(* IEC 61131-3 sources: AXOpen/src/_test/app/SystemConstants, 2 files *)

(* ---- plc_line_IoAddresses.st ---- *)
CONFIGURATION IoAddresses
    VAR_GLOBAL

        // Module rexroth_ctrlx_drive/Inputs
        rexroth_ctrlx_drive_Inputs_P_0_0106_0_0__STO_function__Operating_status_Input AT %IB20 : rexroth_ctrlx_drive_Inputs_P_0_0106_0_0__STO_function__Operating_status_Input_Layout;
        rexroth_ctrlx_drive_Inputs_S_0_0084_0_0__Torque_force_feedback_value_Input AT %IB18 : rexroth_ctrlx_drive_Inputs_S_0_0084_0_0__Torque_force_feedback_value_Input_Layout;
        rexroth_ctrlx_drive_Inputs_S_0_0135_0_0__Drive_status_word__Value_Input AT %IB12 : rexroth_ctrlx_drive_Inputs_S_0_0135_0_0__Drive_status_word__Value_Input_Layout;
        rexroth_ctrlx_drive_Inputs_S_0_0144_0_0__Signal_status_word__Value_Input AT %IB14 : rexroth_ctrlx_drive_Inputs_S_0_0144_0_0__Signal_status_word__Value_Input_Layout;
        rexroth_ctrlx_drive_Inputs_S_0_0386_0_0__Position_controller__Position_actual_value_Input AT %IB0 : rexroth_ctrlx_drive_Inputs_S_0_0386_0_0__Position_controller__Position_actual_value_Input_Layout;
        rexroth_ctrlx_drive_Inputs_S_0_0390_0_0__Diagnostic_message__Manufacturer_status_register_Input AT %IB8 : rexroth_ctrlx_drive_Inputs_S_0_0390_0_0__Diagnostic_message__Manufacturer_status_register_Input_Layout;
        rexroth_ctrlx_drive_Inputs_S_0_0535_0_0__Velocity_controller__Velocity_actual_value_Input AT %IB4 : rexroth_ctrlx_drive_Inputs_S_0_0535_0_0__Velocity_controller__Velocity_actual_value_Input_Layout;
        rexroth_ctrlx_drive_Inputs_S_0_1720_0_2__Power_supply_control__Status_word_Input AT %IB16 : rexroth_ctrlx_drive_Inputs_S_0_1720_0_2__Power_supply_control__Status_word_Input_Layout;

        // Module rexroth_ctrlx_drive/Outputs
        rexroth_ctrlx_drive_Outputs_S_0_0080_0_0__Torque_force_command_value_Output AT %QB24 : rexroth_ctrlx_drive_Outputs_S_0_0080_0_0__Torque_force_command_value_Output_Layout;
        rexroth_ctrlx_drive_Outputs_S_0_0092_0_0__Torque_force_limitation__Limit_value_bipolar_Output AT %QB22 : rexroth_ctrlx_drive_Outputs_S_0_0092_0_0__Torque_force_limitation__Limit_value_bipolar_Output_Layout;
        rexroth_ctrlx_drive_Outputs_S_0_0134_0_0__Master_control_word__Value_Output AT %QB0 : rexroth_ctrlx_drive_Outputs_S_0_0134_0_0__Master_control_word__Value_Output_Layout;
        rexroth_ctrlx_drive_Outputs_S_0_0145_0_0__Signal_control_word__Value_Output AT %QB18 : rexroth_ctrlx_drive_Outputs_S_0_0145_0_0__Signal_control_word__Value_Output_Layout;
        rexroth_ctrlx_drive_Outputs_S_0_0193_0_0__Positioning_jerk_Output AT %QB26 : rexroth_ctrlx_drive_Outputs_S_0_0193_0_0__Positioning_jerk_Output_Layout;
        rexroth_ctrlx_drive_Outputs_S_0_0259_0_0__Positioning_profile__Profile_velocity_Output AT %QB14 : rexroth_ctrlx_drive_Outputs_S_0_0259_0_0__Positioning_profile__Profile_velocity_Output_Layout;
        rexroth_ctrlx_drive_Outputs_S_0_0260_0_0__Positioning_profile__Acceleration_Output AT %QB2 : rexroth_ctrlx_drive_Outputs_S_0_0260_0_0__Positioning_profile__Acceleration_Output_Layout;
        rexroth_ctrlx_drive_Outputs_S_0_0282_0_0__Drive_controlled_positioning__Command_value_Output AT %QB6 : rexroth_ctrlx_drive_Outputs_S_0_0282_0_0__Drive_controlled_positioning__Command_value_Output_Layout;
        rexroth_ctrlx_drive_Outputs_S_0_0359_0_0__Positioning_profile__Deceleration_Output AT %QB10 : rexroth_ctrlx_drive_Outputs_S_0_0359_0_0__Positioning_profile__Deceleration_Output_Layout;
        rexroth_ctrlx_drive_Outputs_S_0_1720_0_1__Power_supply_control__Control_word_Output AT %QB20 : rexroth_ctrlx_drive_Outputs_S_0_1720_0_1__Power_supply_control__Control_word_Output_Layout;
    END_VAR
END_CONFIGURATION

TYPE
    rexroth_ctrlx_drive_Inputs_P_0_0106_0_0__STO_function__Operating_status_Input_Layout : STRUCT
        Signals_0 AT %B0 : WORD;
    END_STRUCT;
END_TYPE

TYPE
    rexroth_ctrlx_drive_Inputs_S_0_0084_0_0__Torque_force_feedback_value_Input_Layout : STRUCT
        Signals_0 AT %B0 : INT;
    END_STRUCT;
END_TYPE

TYPE
    rexroth_ctrlx_drive_Inputs_S_0_0135_0_0__Drive_status_word__Value_Input_Layout : STRUCT
        Signals_0 AT %X0.3 : BOOL;
        Signals_1 AT %X0.4 : BOOL;
        Signals_2 AT %X0.5 : BOOL;
        Signals_3 AT %X0.7 : BOOL;
        Signals_4 AT %X1.0 : BOOL;
        Signals_5 AT %X1.1 : BOOL;
        Signals_6 AT %X1.2 : BOOL;
        Signals_7 AT %X1.4 : BOOL;
        Signals_8 AT %X1.5 : BOOL;
        Signals_9 AT %X1.6 : BOOL;
        Signals_10 AT %X1.7 : BOOL;
    END_STRUCT;
END_TYPE

TYPE
    rexroth_ctrlx_drive_Inputs_S_0_0144_0_0__Signal_status_word__Value_Input_Layout : STRUCT
        Signals_0 AT %B0 : WORD;
    END_STRUCT;
END_TYPE

TYPE
    rexroth_ctrlx_drive_Inputs_S_0_0386_0_0__Position_controller__Position_actual_value_Input_Layout : STRUCT
        Signals_0 AT %B0 : DINT;
    END_STRUCT;
END_TYPE

TYPE
    rexroth_ctrlx_drive_Inputs_S_0_0390_0_0__Diagnostic_message__Manufacturer_status_register_Input_Layout : STRUCT
        Signals_0 AT %B0 : DWORD;
    END_STRUCT;
END_TYPE

TYPE
    rexroth_ctrlx_drive_Inputs_S_0_0535_0_0__Velocity_controller__Velocity_actual_value_Input_Layout : STRUCT
        Signals_0 AT %B0 : DINT;
    END_STRUCT;
END_TYPE

TYPE
    rexroth_ctrlx_drive_Inputs_S_0_1720_0_2__Power_supply_control__Status_word_Input_Layout : STRUCT
        Signals_0 AT %B0 : WORD;
    END_STRUCT;
END_TYPE

TYPE
    rexroth_ctrlx_drive_Outputs_S_0_0080_0_0__Torque_force_command_value_Output_Layout : STRUCT
        Signals_0 AT %B0 : INT;
    END_STRUCT;
END_TYPE

TYPE
    rexroth_ctrlx_drive_Outputs_S_0_0092_0_0__Torque_force_limitation__Limit_value_bipolar_Output_Layout : STRUCT
        Signals_0 AT %B0 : WORD;
    END_STRUCT;
END_TYPE

TYPE
    rexroth_ctrlx_drive_Outputs_S_0_0134_0_0__Master_control_word__Value_Output_Layout : STRUCT
        Signals_0 AT %X1.0 : BOOL;
        Signals_1 AT %X1.1 : BOOL;
        Signals_2 AT %X1.2 : BOOL;
        Signals_3 AT %X1.5 : BOOL;
        Signals_4 AT %X1.6 : BOOL;
        Signals_5 AT %X1.7 : BOOL;
    END_STRUCT;
END_TYPE

TYPE
    rexroth_ctrlx_drive_Outputs_S_0_0145_0_0__Signal_control_word__Value_Output_Layout : STRUCT
        Signals_0 AT %B0 : WORD;
    END_STRUCT;
END_TYPE

TYPE
    rexroth_ctrlx_drive_Outputs_S_0_0193_0_0__Positioning_jerk_Output_Layout : STRUCT
        Signals_0 AT %B0 : DINT;
    END_STRUCT;
END_TYPE

TYPE
    rexroth_ctrlx_drive_Outputs_S_0_0259_0_0__Positioning_profile__Profile_velocity_Output_Layout : STRUCT
        Signals_0 AT %B0 : DWORD;
    END_STRUCT;
END_TYPE

TYPE
    rexroth_ctrlx_drive_Outputs_S_0_0260_0_0__Positioning_profile__Acceleration_Output_Layout : STRUCT
        Signals_0 AT %B0 : DINT;
    END_STRUCT;
END_TYPE

TYPE
    rexroth_ctrlx_drive_Outputs_S_0_0282_0_0__Drive_controlled_positioning__Command_value_Output_Layout : STRUCT
        Signals_0 AT %B0 : DINT;
    END_STRUCT;
END_TYPE

TYPE
    rexroth_ctrlx_drive_Outputs_S_0_0359_0_0__Positioning_profile__Deceleration_Output_Layout : STRUCT
        Signals_0 AT %B0 : DINT;
    END_STRUCT;
END_TYPE

TYPE
    rexroth_ctrlx_drive_Outputs_S_0_1720_0_1__Power_supply_control__Control_word_Output_Layout : STRUCT
        Signals_0 AT %B0 : WORD;
    END_STRUCT;
END_TYPE

(* ---- plc_line_HwIdentifiers.st ---- *)
CONFIGURATION HardwareIDs
    VAR_GLOBAL CONSTANT
        plc_line_HwID : UINT := UINT#32;
        plc_line_Rail_0_HwID : UINT := UINT#284;
        plc_line_plc_line_HwID : UINT := UINT#48;
        plc_line_plc_line_CPU_display_1_HwID : UINT := UINT#54;
        plc_line_plc_line_Card_reader_writer_1_HwID : UINT := UINT#51;
        plc_line_plc_line_DP_interface_1_HwID : UINT := UINT#60;
        plc_line_plc_line_OPC_UA_1_HwID : UINT := UINT#117;
        plc_line_plc_line_PROFINET_interface_1_HwID : UINT := UINT#64;
        plc_line_plc_line_PROFINET_interface_1_Port_1_HwID : UINT := UINT#65;
        plc_line_plc_line_PROFINET_interface_1_Port_2_HwID : UINT := UINT#66;
        plc_line_plc_line_PROFINET_interface_2_HwID : UINT := UINT#72;
        plc_line_plc_line_PROFINET_interface_2_Port_3_HwID : UINT := UINT#73;
        plc_line_plc_line_Virtual_communication_interface_HwID : UINT := UINT#135;
        profinet_plc_line_HwID : UINT := UINT#256;
        rexroth_ctrlx_drive_HwID : UINT := UINT#258;
        rexroth_ctrlx_drive_Inputs_HwID : UINT := UINT#264;
        rexroth_ctrlx_drive_Outputs_HwID : UINT := UINT#263;
        rexroth_ctrlx_drive_P_0_0106_0_0__STO_function__Operating_status_HwID : UINT := UINT#272;
        rexroth_ctrlx_drive_Rack_HwID : UINT := UINT#261;
        rexroth_ctrlx_drive_S_0_0080_0_0__Torque_force_command_value_HwID : UINT := UINT#281;
        rexroth_ctrlx_drive_S_0_0084_0_0__Torque_force_feedback_value_HwID : UINT := UINT#271;
        rexroth_ctrlx_drive_S_0_0092_0_0__Torque_force_limitation__Limit_value_bipolar_HwID : UINT := UINT#280;
        rexroth_ctrlx_drive_S_0_0134_0_0__Master_control_word__Value_HwID : UINT := UINT#273;
        rexroth_ctrlx_drive_S_0_0135_0_0__Drive_status_word__Value_HwID : UINT := UINT#268;
        rexroth_ctrlx_drive_S_0_0144_0_0__Signal_status_word__Value_HwID : UINT := UINT#269;
        rexroth_ctrlx_drive_S_0_0145_0_0__Signal_control_word__Value_HwID : UINT := UINT#278;
        rexroth_ctrlx_drive_S_0_0193_0_0__Positioning_jerk_HwID : UINT := UINT#282;
        rexroth_ctrlx_drive_S_0_0259_0_0__Positioning_profile__Profile_velocity_HwID : UINT := UINT#277;
        rexroth_ctrlx_drive_S_0_0260_0_0__Positioning_profile__Acceleration_HwID : UINT := UINT#274;
        rexroth_ctrlx_drive_S_0_0282_0_0__Drive_controlled_positioning__Command_value_HwID : UINT := UINT#275;
        rexroth_ctrlx_drive_S_0_0359_0_0__Positioning_profile__Deceleration_HwID : UINT := UINT#276;
        rexroth_ctrlx_drive_S_0_0386_0_0__Position_controller__Position_actual_value_HwID : UINT := UINT#265;
        rexroth_ctrlx_drive_S_0_0390_0_0__Diagnostic_message__Manufacturer_status_register_HwID : UINT := UINT#267;
        rexroth_ctrlx_drive_S_0_0535_0_0__Velocity_controller__Velocity_actual_value_HwID : UINT := UINT#266;
        rexroth_ctrlx_drive_S_0_1720_0_1__Power_supply_control__Control_word_HwID : UINT := UINT#279;
        rexroth_ctrlx_drive_S_0_1720_0_2__Power_supply_control__Status_word_HwID : UINT := UINT#270;
        rexroth_ctrlx_drive_rexroth_ctrlx_drive_HwID : UINT := UINT#262;
        rexroth_ctrlx_drive_rexroth_ctrlx_drive_XCS_interface_PF30_HwID : UINT := UINT#257;
        rexroth_ctrlx_drive_rexroth_ctrlx_drive_XCS_interface_PF30_Port_1_HwID : UINT := UINT#259;
        rexroth_ctrlx_drive_rexroth_ctrlx_drive_XCS_interface_PF30_Port_2_HwID : UINT := UINT#260;
        rexroth_ctrlx_drive_rexroth_ctrlx_drive_ctrlX_DRIVE_XCS_HwID : UINT := UINT#283;

    END_VAR
END_CONFIGURATION
